{attribute 'GeneratedUsingTerminal: EP3744-0041-0016'}
{attribute addProperty BoxType "EP3744-0041-0016"}
{attribute addProperty Id "OutputAT %Q*ARRAY[0..1] OF BOOL2"}
{attribute addProperty CRC "2036329114"}
{attribute addProperty Size "2"}
TYPE DIG_Outputs_DE230DD5 :
STRUCT
	{attribute addProperty Name "Output"}
	Output AT %Q* : ARRAY[0..1] OF BOOL;
END_STRUCT
END_TYPE

(* stored: Version 1.2.0.0, ProductVersion 3.1.4024.9
   DUT DIG_Outputs_DE230DD5: Id {8069d4aa-9ac4-4b95-8916-4a6cb974deb8} *)
